(* PLC project pi@codesys.project, CODESYS CODESYS V3.5 SP12 *)
(* stored: creationDateTime 2018-04-12T11:06:56.1462024, modificationDateTime 2018-04-12T11:06:35.882732 *)

{attribute 'qualified_only'}
{attribute 'strict'}
TYPE DUT_ENUM :
(
	enum_member := 0
);
END_TYPE

TYPE SPINDLE_STRUCT :
STRUCT
	none:			 INT := 0;
	ace_v1:			 INT := 1;
	ace_v2:			 INT := 2;
	ace_v3:			 INT := 3;
	ace_v4:			 INT := 4;
	hgvuz_v1:		 INT := 5;
	vakuum_v2:		 INT := 6;
	frontspann_v1:	 INT := 7;
	universal_v1:	 INT := 8;
	achsklemmung_v1: INT := 9;
	ahk_v1:			 INT := 10;
END_STRUCT
END_TYPE

TYPE DUT_ALIAS : BOOL; END_TYPE

{attribute 'qualified_only'}
{attribute 'strict'}
TYPE SPINDLE :
(
	None			 := 0,
	ace_v1			 := 1,
	ace_v2			 := 2,
	ace_v3			 := 3,
	ace_v4			 := 4,
	hgvuz_v1		 := 5,
	vakuum_v2		 := 6,
	frontspann_v1	 := 7,
	universal_v1	 := 8,
	achsklemmung_v1	 := 9,
	ahk_v1			 := 10
) := None;
END_TYPE

{attribute 'qualified_only'}
{attribute 'strict'}
TYPE TELEGRAM :
(
	NONE := '',
	BRAKE_RELEASE := 'br$$$$0',
	BRAKE_APPLY := 'br$$$$1',
	BRAKE_STATUS := 'cs§§'
)STRING;
END_TYPE

TYPE udtInput : 
STRUCT
	S2: BOOL;		// Adapter check
	S3: BOOL;		// Mazak ACE
	SIX: BOOL;		// Micro-switch spindle index
	OT_SB2: BOOL;	// One-hand control handle: 1st button
	OT_SB3: BOOL;	// One-hand control handle: 2nd button
	KeySw_S2: BOOL;	// Key switch
	
END_STRUCT
END_TYPE

TYPE udtOutput :
STRUCT
	_4Y0 : BOOL; // ACE_V1/V4 = SITEMA
	_4Y1 : BOOL; // ACE_V1/V4 = KLAUEN
	_4Y2 : BOOL; // Bremse
	_4Y3 : BOOL; // Index
END_STRUCT
END_TYPE

PROGRAM PLC_PRG
VAR
	temp: BOOL;
	i: INT;
	dummy1 : INT;
	dummy2 : INT;
	instEject: Eject;
	
END_VAR

                    i := i + 1;
IF i MOD (dummy1 * 10) = 0 THEN
	%QB0 := %QB0 +1;
END_IF
IF i MOD (dummy2 * 10) = 0 THEN
	%QB1 := %QB1 - 1;	
END_If



Modbus_TCP_Master.uiConnectedSlaves;
Modbus_TCP_Master.xSlaveError;
Modbus_TCP_Master.xStop;

//Modbus_TCP_Slave.byModbusError;
//Modbus_TCP_Slave.ComSettings;
//Modbus_TCP_Slave.ComState;
//Modbus_TCP_Slave.iChannelIndex;

instEject(locked := temp,
	);


                  
END_PROGRAM

FUNCTION_BLOCK KOP
VAR_INPUT
END_VAR
VAR_OUTPUT
END_VAR
VAR
END_VAR

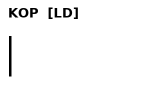
(* LD diagram, written out as Structured Text *)
(* --- network --- *)
END_FUNCTION_BLOCK

FUNCTION_BLOCK FUP
VAR_INPUT
END_VAR
VAR_OUTPUT
END_VAR
VAR
END_VAR

(* FBD diagram, written out as Structured Text *)
END_FUNCTION_BLOCK

FUNCTION_BLOCK Eject
VAR_INPUT
	spindleType : INT;
	
END_VAR
VAR_OUTPUT
	_4Y0: BOOL;
	_4Y1: BOOL;
	response: STRING(10);
END_VAR
VAR
	ejectStartStop: BOOL;
	toolActive: BOOL;
	ejectActive: BOOL;
	
END_VAR
VAR_IN_OUT
	locked: BOOL;
END_VAR
VAR CONSTANT
	TIME18: TIME := T#4000MS;
	TIME19: TIME := T#200MS;
	TIME20: TIME := T#3000MS;
	TIME21: TIME := T#400MS;
	TIME22: TIME := T#4000MS;
	TIME25: TIME := T#3000MS;
END_VAR

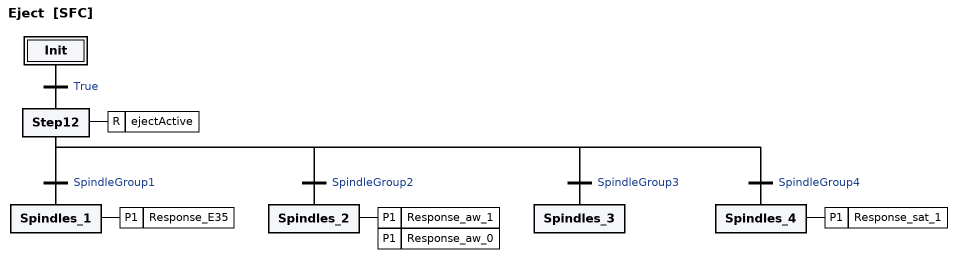
INITIAL_STEP Init:
END_STEP
TRANSITION FROM Init TO Step12
  := True;
END_TRANSITION
STEP Step12:
  ejectActive(R);
END_STEP
TRANSITION FROM Step12 TO Spindles_1
  := SpindleGroup1;
END_TRANSITION
TRANSITION FROM Step12 TO Spindles_2
  := SpindleGroup2;
END_TRANSITION
TRANSITION FROM Step12 TO Spindles_3
  := SpindleGroup3;
END_TRANSITION
TRANSITION FROM Step12 TO Spindles_4
  := SpindleGroup4;
END_TRANSITION
STEP Spindles_1:
  Response_E35(P1);
END_STEP
STEP Spindles_2:
  Response_aw_1(P1);
  Response_aw_0(P1);
END_STEP
STEP Spindles_3:
END_STEP
STEP Spindles_4:
  Response_sat_1(P1);
END_STEP

ACTION Response_E35:
                        response := 'aw$$$$1E35';
                      
END_ACTION

ACTION Response_aw_1:
                        response := 'aw$$$$1';
                      
END_ACTION

ACTION Response_aw_0:
                        response := 'aw$$$$0';
                      
END_ACTION

ACTION Response_sat_1:
                        response := 'sat$$1';
                      
END_ACTION
END_FUNCTION_BLOCK

FUNCTION_BLOCK CFC
VAR_INPUT
END_VAR
VAR_OUTPUT
END_VAR
VAR
END_VAR

(* CFC diagram, written out as Structured Text *)
END_FUNCTION_BLOCK

FUNCTION_BLOCK SpindleBrake
VAR_INPUT
	spindleType: BOOL; // Spindle type
	telegramCtrl: STRING; // Control telegram
	buttonCtrl: BOOL; // Control button
END_VAR
VAR_OUTPUT
	_4Y2: BOOL; // Spindle brake valve
	ledOff: BOOL; // 
	ledOn: BOOL;
	telegramSts: STRING; // Status telegram
END_VAR
VAR
END_VAR

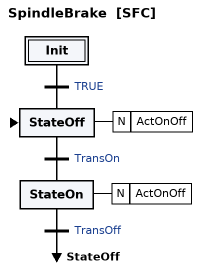
INITIAL_STEP Init:
END_STEP
TRANSITION FROM Init TO StateOff
  := TRUE;
END_TRANSITION
STEP StateOff:
  ActOnOff(N);
END_STEP
TRANSITION FROM StateOff TO StateOn
  := TransOn;
END_TRANSITION
STEP StateOn:
  ActOnOff(N);
END_STEP
TRANSITION FROM StateOn TO StateOff
  := TransOff;
END_TRANSITION

ACTION ActOnOff:
                        _4Y2 := StateOn.x;
ledOff := StateOff.x;
ledOn := StateOn.x;

IF StateOff._x THEN
	telegramSts := TELEGRAM.BRAKE_RELEASE;
ELSIF StateOn._x THEN
	telegramSts := TELEGRAM.BRAKE_APPLY;
ELSE
	telegramSts := TELEGRAM.NONE;
END_IF

//IF telegramCtrl = TELEGRAM.BRAKE_STATUS THEN
//	telegramSts := TELEGRAM.NONE;
//	IF StepOff.x THEN
//		telegramSts := 'cs§§0';
//	ELSIF StepOn.x THEN
//		telegramSts := 'cs§§1';
//	END_IF
//END_IF
                      
END_ACTION
END_FUNCTION_BLOCK

FUNCTION_BLOCK OutputMapping
VAR_INPUT
	out : udtOutput;
	cfg : INT;
END_VAR
VAR_OUTPUT
	dq : ARRAY [0..1, 0..7] OF BOOL;
	
END_VAR
VAR
	dq0 AT %Q*: BOOL;
END_VAR

                    dq[0, 0] := out._4Y0;
dq[0, 1] := out._4Y1;
dq[0, 2] := out._4Y2;
dq[0, 3] := out._4Y3;

dq0 := TRue;
                  
END_FUNCTION_BLOCK

FUNCTION_BLOCK Keypad
VAR_INPUT
END_VAR
VAR_OUTPUT
END_VAR
VAR
	disable: BOOL := FALSE;
END_VAR

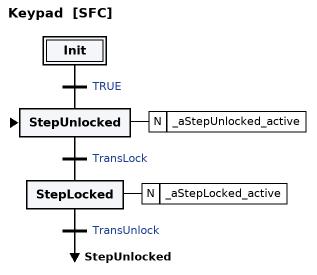
INITIAL_STEP Init:
END_STEP
TRANSITION FROM Init TO StepUnlocked
  := TRUE;
END_TRANSITION
STEP StepUnlocked:
  _aStepUnlocked_active(N);
END_STEP
TRANSITION FROM StepUnlocked TO StepLocked
  := TransLock;
END_TRANSITION
STEP StepLocked:
  _aStepLocked_active(N);
END_STEP
TRANSITION FROM StepLocked TO StepUnlocked
  := TransUnlock;
END_TRANSITION

ACTION _aStepUnlocked_active:
                        // TODO
                      
END_ACTION

ACTION _aStepLocked_active:
                        // TODO

                      
END_ACTION
END_FUNCTION_BLOCK

FUNCTION_BLOCK InputMapping
VAR_INPUT
	di : ARRAY [0..1, 0..7] OF BOOL;
	cfg : INT;
END_VAR
VAR_IN_OUT
	in : udtInput;
END_VAR

                    in.S2 := di[0, 2];
in.S3 := di[0, 3];
                  
END_FUNCTION_BLOCK

PROGRAM POU
VAR
	instKeypad: Keypad;
END_VAR

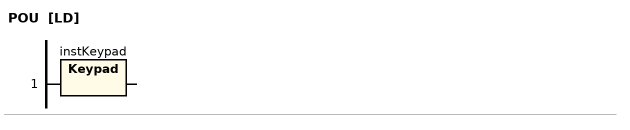
(* LD diagram, written out as Structured Text *)

instKeypad();
END_PROGRAM

CONFIGURATION Device
  RESOURCE Application ON PLC
(* global variable list GVL *)
{attribute 'qualified_only'}
VAR_GLOBAL
	di : ARRAY[0..1, 0..7] OF BOOL;
	_4Y0: BOOL;
	in : udtInput;
	out : udtOutput;
	testBool : BOOL;
	
END_VAR
(* global variable list PersistentVars *)
{attribute 'qualified_only'}
VAR_GLOBAL PERSISTENT RETAIN
END_VAR
(* global variable list GVL_1 *)
{attribute 'qualified_only'}
VAR_CONFIG
	
END_VAR
    TASK MainTask(INTERVAL := T#4ms, PRIORITY := 1);
    PROGRAM PLC_PRG WITH MainTask : PLC_PRG;
    PROGRAM POU WITH MainTask : POU;
  END_RESOURCE
END_CONFIGURATION

CONFIGURATION Ethernet_1
END_CONFIGURATION

CONFIGURATION Modbus_TCP_Master
END_CONFIGURATION

CONFIGURATION Modbus_TCP_Slave
END_CONFIGURATION

CONFIGURATION Ethernet
END_CONFIGURATION

CONFIGURATION ModbusTCP_Slave_Device
END_CONFIGURATION

CONFIGURATION SoftMotion General Axis Pool
END_CONFIGURATION

CONFIGURATION I²C
END_CONFIGURATION

CONFIGURATION I2C_master
END_CONFIGURATION

CONFIGURATION I2HE_Digital_Inputs_IO_driver_1
END_CONFIGURATION

CONFIGURATION I2HE_Digital_Inputs_IO_driver_2
END_CONFIGURATION

CONFIGURATION I2HA_Digital_Outputs_IO_driver_1
END_CONFIGURATION

CONFIGURATION I2HA_Digital_Outputs_IO_driver_2
END_CONFIGURATION

CONFIGURATION SPI
END_CONFIGURATION

CONFIGURATION GPIOs_A_B
END_CONFIGURATION

CONFIGURATION Onewire
END_CONFIGURATION

CONFIGURATION Camera device
END_CONFIGURATION

CONFIGURATION <Leer>
END_CONFIGURATION
